TYPE TFMachinePalletizer_WorkAreaSort :
STRUCT
	Distance : LREAL;
	cwa : UINT;
END_STRUCT
END_TYPE

(* stored: Version 1.1.0.1, ProductVersion 3.1.4024.11
   DUT TFMachinePalletizer_WorkAreaSort: Id {27ed1585-73b5-43d7-81f2-ac1f8192413a} *)
